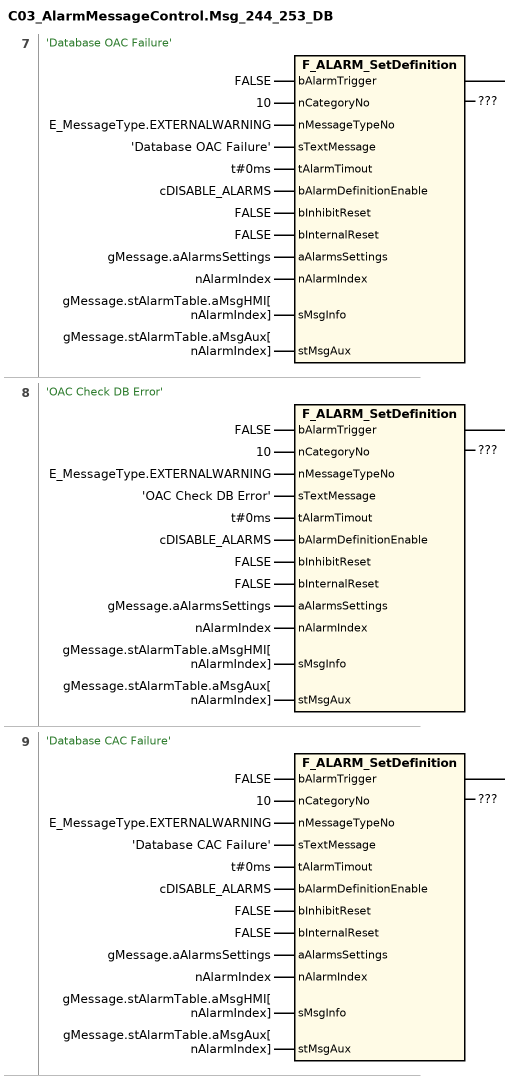
// NETWORK 7
// 'Database OAC Failure'
F_ALARM_SetDefinition(bAlarmTrigger := FALSE, nCategoryNo := 10, nMessageTypeNo := E_MessageType.EXTERNALWARNING, sTextMessage := 'Database OAC Failure', tAlarmTimout := t#0ms, bAlarmDefinitionEnable := cDISABLE_ALARMS, bInhibitReset := FALSE, bInternalReset := FALSE, aAlarmsSettings := gMessage.aAlarmsSettings, nAlarmIndex := nAlarmIndex, sMsgInfo := gMessage.stAlarmTable.aMsgHMI[nAlarmIndex], stMsgAux := gMessage.stAlarmTable.aMsgAux[nAlarmIndex]);

// NETWORK 8
// 'OAC Check DB Error'
F_ALARM_SetDefinition(bAlarmTrigger := FALSE, nCategoryNo := 10, nMessageTypeNo := E_MessageType.EXTERNALWARNING, sTextMessage := 'OAC Check DB Error', tAlarmTimout := t#0ms, bAlarmDefinitionEnable := cDISABLE_ALARMS, bInhibitReset := FALSE, bInternalReset := FALSE, aAlarmsSettings := gMessage.aAlarmsSettings, nAlarmIndex := nAlarmIndex, sMsgInfo := gMessage.stAlarmTable.aMsgHMI[nAlarmIndex], stMsgAux := gMessage.stAlarmTable.aMsgAux[nAlarmIndex]);

// NETWORK 9
// 'Database CAC Failure'
F_ALARM_SetDefinition(bAlarmTrigger := FALSE, nCategoryNo := 10, nMessageTypeNo := E_MessageType.EXTERNALWARNING, sTextMessage := 'Database CAC Failure', tAlarmTimout := t#0ms, bAlarmDefinitionEnable := cDISABLE_ALARMS, bInhibitReset := FALSE, bInternalReset := FALSE, aAlarmsSettings := gMessage.aAlarmsSettings, nAlarmIndex := nAlarmIndex, sMsgInfo := gMessage.stAlarmTable.aMsgHMI[nAlarmIndex], stMsgAux := gMessage.stAlarmTable.aMsgAux[nAlarmIndex]);

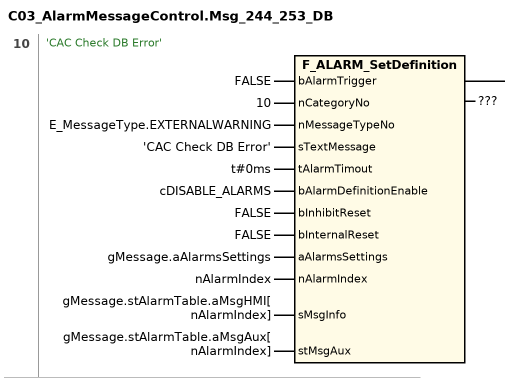
// NETWORK 10
// 'CAC Check DB Error'
F_ALARM_SetDefinition(bAlarmTrigger := FALSE, nCategoryNo := 10, nMessageTypeNo := E_MessageType.EXTERNALWARNING, sTextMessage := 'CAC Check DB Error', tAlarmTimout := t#0ms, bAlarmDefinitionEnable := cDISABLE_ALARMS, bInhibitReset := FALSE, bInternalReset := FALSE, aAlarmsSettings := gMessage.aAlarmsSettings, nAlarmIndex := nAlarmIndex, sMsgInfo := gMessage.stAlarmTable.aMsgHMI[nAlarmIndex], stMsgAux := gMessage.stAlarmTable.aMsgAux[nAlarmIndex]);
END_ACTION

ACTION Msg_254_255_Reserved:
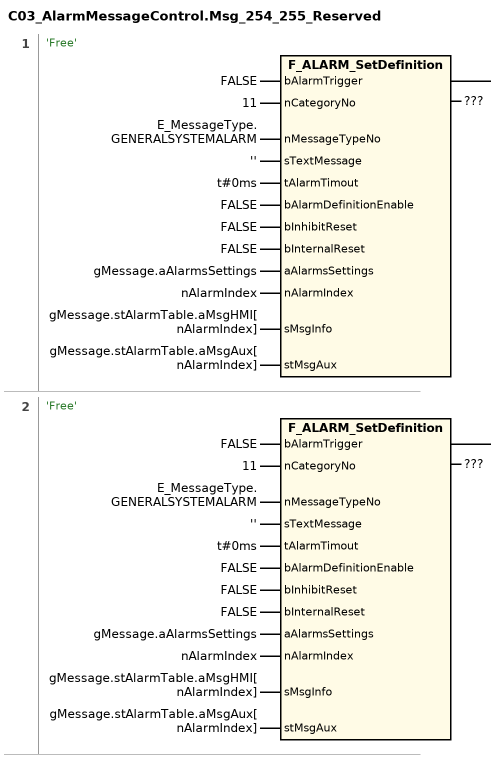
// NETWORK 1
// 'Free'
F_ALARM_SetDefinition(bAlarmTrigger := FALSE, nCategoryNo := 11, nMessageTypeNo := E_MessageType.GENERALSYSTEMALARM, sTextMessage := '', tAlarmTimout := t#0ms, bAlarmDefinitionEnable := FALSE, bInhibitReset := FALSE, bInternalReset := FALSE, aAlarmsSettings := gMessage.aAlarmsSettings, nAlarmIndex := nAlarmIndex, sMsgInfo := gMessage.stAlarmTable.aMsgHMI[nAlarmIndex], stMsgAux := gMessage.stAlarmTable.aMsgAux[nAlarmIndex]);

// NETWORK 2
// 'Free'
F_ALARM_SetDefinition(bAlarmTrigger := FALSE, nCategoryNo := 11, nMessageTypeNo := E_MessageType.GENERALSYSTEMALARM, sTextMessage := '', tAlarmTimout := t#0ms, bAlarmDefinitionEnable := FALSE, bInhibitReset := FALSE, bInternalReset := FALSE, aAlarmsSettings := gMessage.aAlarmsSettings, nAlarmIndex := nAlarmIndex, sMsgInfo := gMessage.stAlarmTable.aMsgHMI[nAlarmIndex], stMsgAux := gMessage.stAlarmTable.aMsgAux[nAlarmIndex]);
END_ACTION

ACTION MsgReset:
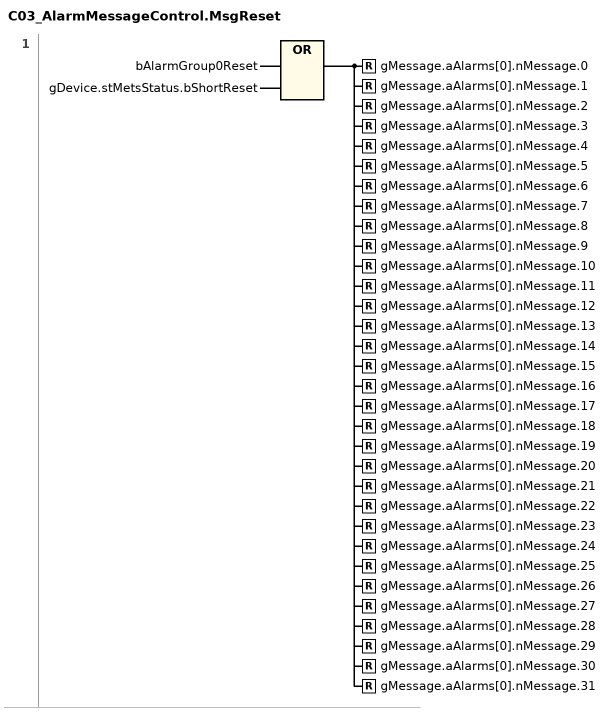
// NETWORK 1
_w1 := bAlarmGroup0Reset OR gDevice.stMetsStatus.bShortReset;
gMessage.aAlarms[0].nMessage.0 R= _w1;
gMessage.aAlarms[0].nMessage.1 R= _w1;
gMessage.aAlarms[0].nMessage.2 R= _w1;
gMessage.aAlarms[0].nMessage.3 R= _w1;
gMessage.aAlarms[0].nMessage.4 R= _w1;
gMessage.aAlarms[0].nMessage.5 R= _w1;
gMessage.aAlarms[0].nMessage.6 R= _w1;
gMessage.aAlarms[0].nMessage.7 R= _w1;
gMessage.aAlarms[0].nMessage.8 R= _w1;
gMessage.aAlarms[0].nMessage.9 R= _w1;
gMessage.aAlarms[0].nMessage.10 R= _w1;
gMessage.aAlarms[0].nMessage.11 R= _w1;
gMessage.aAlarms[0].nMessage.12 R= _w1;
gMessage.aAlarms[0].nMessage.13 R= _w1;
gMessage.aAlarms[0].nMessage.14 R= _w1;
gMessage.aAlarms[0].nMessage.15 R= _w1;
gMessage.aAlarms[0].nMessage.16 R= _w1;
gMessage.aAlarms[0].nMessage.17 R= _w1;
gMessage.aAlarms[0].nMessage.18 R= _w1;
gMessage.aAlarms[0].nMessage.19 R= _w1;
gMessage.aAlarms[0].nMessage.20 R= _w1;
gMessage.aAlarms[0].nMessage.21 R= _w1;
gMessage.aAlarms[0].nMessage.22 R= _w1;
gMessage.aAlarms[0].nMessage.23 R= _w1;
gMessage.aAlarms[0].nMessage.24 R= _w1;
gMessage.aAlarms[0].nMessage.25 R= _w1;
gMessage.aAlarms[0].nMessage.26 R= _w1;
gMessage.aAlarms[0].nMessage.27 R= _w1;
gMessage.aAlarms[0].nMessage.28 R= _w1;
gMessage.aAlarms[0].nMessage.29 R= _w1;
gMessage.aAlarms[0].nMessage.30 R= _w1;
gMessage.aAlarms[0].nMessage.31 R= _w1;

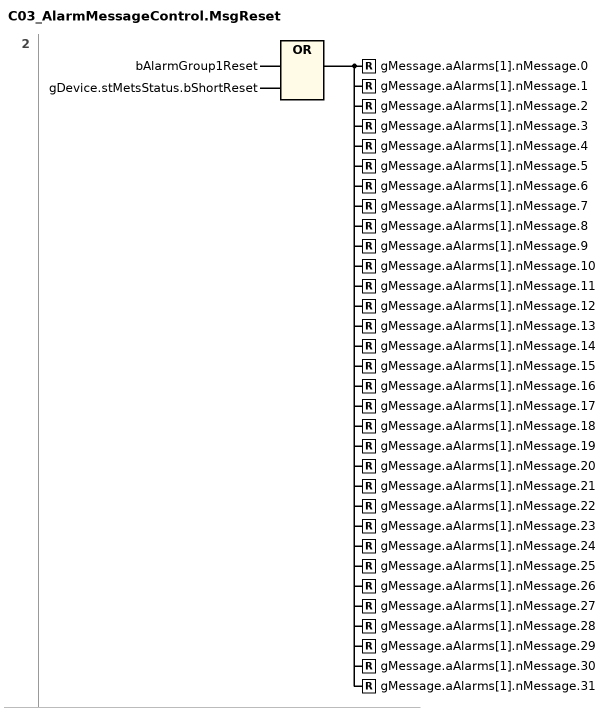
// NETWORK 2
_w2 := bAlarmGroup1Reset OR gDevice.stMetsStatus.bShortReset;
gMessage.aAlarms[1].nMessage.0 R= _w2;
gMessage.aAlarms[1].nMessage.1 R= _w2;
gMessage.aAlarms[1].nMessage.2 R= _w2;
gMessage.aAlarms[1].nMessage.3 R= _w2;
gMessage.aAlarms[1].nMessage.4 R= _w2;
gMessage.aAlarms[1].nMessage.5 R= _w2;
gMessage.aAlarms[1].nMessage.6 R= _w2;
gMessage.aAlarms[1].nMessage.7 R= _w2;
gMessage.aAlarms[1].nMessage.8 R= _w2;
gMessage.aAlarms[1].nMessage.9 R= _w2;
gMessage.aAlarms[1].nMessage.10 R= _w2;
gMessage.aAlarms[1].nMessage.11 R= _w2;
gMessage.aAlarms[1].nMessage.12 R= _w2;
gMessage.aAlarms[1].nMessage.13 R= _w2;
gMessage.aAlarms[1].nMessage.14 R= _w2;
gMessage.aAlarms[1].nMessage.15 R= _w2;
gMessage.aAlarms[1].nMessage.16 R= _w2;
gMessage.aAlarms[1].nMessage.17 R= _w2;
gMessage.aAlarms[1].nMessage.18 R= _w2;
gMessage.aAlarms[1].nMessage.19 R= _w2;
gMessage.aAlarms[1].nMessage.20 R= _w2;
gMessage.aAlarms[1].nMessage.21 R= _w2;
gMessage.aAlarms[1].nMessage.22 R= _w2;
gMessage.aAlarms[1].nMessage.23 R= _w2;
gMessage.aAlarms[1].nMessage.24 R= _w2;
gMessage.aAlarms[1].nMessage.25 R= _w2;
gMessage.aAlarms[1].nMessage.26 R= _w2;
gMessage.aAlarms[1].nMessage.27 R= _w2;
gMessage.aAlarms[1].nMessage.28 R= _w2;
gMessage.aAlarms[1].nMessage.29 R= _w2;
gMessage.aAlarms[1].nMessage.30 R= _w2;
gMessage.aAlarms[1].nMessage.31 R= _w2;

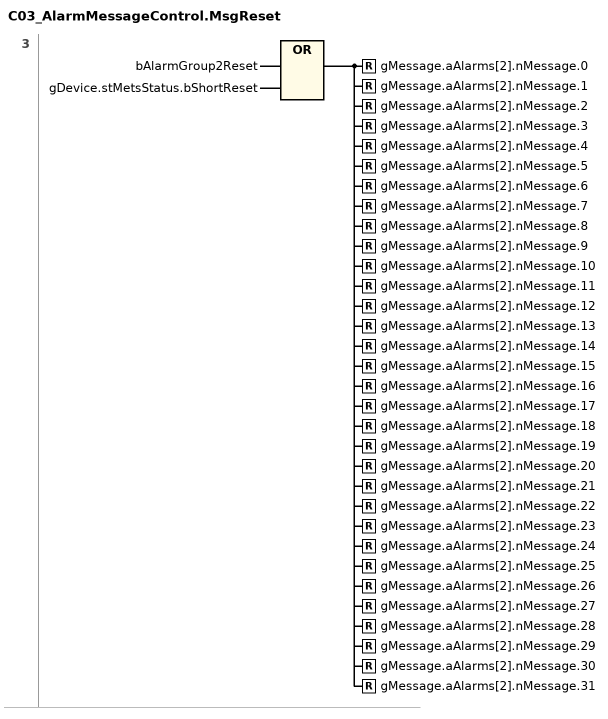
// NETWORK 3
_w3 := bAlarmGroup2Reset OR gDevice.stMetsStatus.bShortReset;
gMessage.aAlarms[2].nMessage.0 R= _w3;
gMessage.aAlarms[2].nMessage.1 R= _w3;
gMessage.aAlarms[2].nMessage.2 R= _w3;
gMessage.aAlarms[2].nMessage.3 R= _w3;
gMessage.aAlarms[2].nMessage.4 R= _w3;
gMessage.aAlarms[2].nMessage.5 R= _w3;
gMessage.aAlarms[2].nMessage.6 R= _w3;
gMessage.aAlarms[2].nMessage.7 R= _w3;
gMessage.aAlarms[2].nMessage.8 R= _w3;
gMessage.aAlarms[2].nMessage.9 R= _w3;
gMessage.aAlarms[2].nMessage.10 R= _w3;
gMessage.aAlarms[2].nMessage.11 R= _w3;
gMessage.aAlarms[2].nMessage.12 R= _w3;
gMessage.aAlarms[2].nMessage.13 R= _w3;
gMessage.aAlarms[2].nMessage.14 R= _w3;
gMessage.aAlarms[2].nMessage.15 R= _w3;
gMessage.aAlarms[2].nMessage.16 R= _w3;
gMessage.aAlarms[2].nMessage.17 R= _w3;
gMessage.aAlarms[2].nMessage.18 R= _w3;
gMessage.aAlarms[2].nMessage.19 R= _w3;
gMessage.aAlarms[2].nMessage.20 R= _w3;
gMessage.aAlarms[2].nMessage.21 R= _w3;
gMessage.aAlarms[2].nMessage.22 R= _w3;
gMessage.aAlarms[2].nMessage.23 R= _w3;
gMessage.aAlarms[2].nMessage.24 R= _w3;
gMessage.aAlarms[2].nMessage.25 R= _w3;
gMessage.aAlarms[2].nMessage.26 R= _w3;
gMessage.aAlarms[2].nMessage.27 R= _w3;
gMessage.aAlarms[2].nMessage.28 R= _w3;
gMessage.aAlarms[2].nMessage.29 R= _w3;
gMessage.aAlarms[2].nMessage.30 R= _w3;
gMessage.aAlarms[2].nMessage.31 R= _w3;

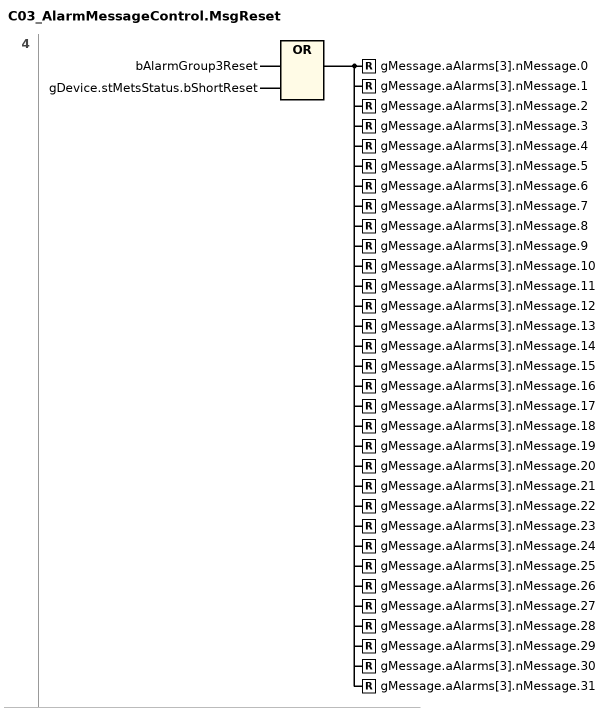
// NETWORK 4
_w4 := bAlarmGroup3Reset OR gDevice.stMetsStatus.bShortReset;
gMessage.aAlarms[3].nMessage.0 R= _w4;
gMessage.aAlarms[3].nMessage.1 R= _w4;
gMessage.aAlarms[3].nMessage.2 R= _w4;
gMessage.aAlarms[3].nMessage.3 R= _w4;
gMessage.aAlarms[3].nMessage.4 R= _w4;
gMessage.aAlarms[3].nMessage.5 R= _w4;
gMessage.aAlarms[3].nMessage.6 R= _w4;
gMessage.aAlarms[3].nMessage.7 R= _w4;
gMessage.aAlarms[3].nMessage.8 R= _w4;
gMessage.aAlarms[3].nMessage.9 R= _w4;
gMessage.aAlarms[3].nMessage.10 R= _w4;
gMessage.aAlarms[3].nMessage.11 R= _w4;
gMessage.aAlarms[3].nMessage.12 R= _w4;
gMessage.aAlarms[3].nMessage.13 R= _w4;
gMessage.aAlarms[3].nMessage.14 R= _w4;
gMessage.aAlarms[3].nMessage.15 R= _w4;
gMessage.aAlarms[3].nMessage.16 R= _w4;
gMessage.aAlarms[3].nMessage.17 R= _w4;
gMessage.aAlarms[3].nMessage.18 R= _w4;
gMessage.aAlarms[3].nMessage.19 R= _w4;
gMessage.aAlarms[3].nMessage.20 R= _w4;
gMessage.aAlarms[3].nMessage.21 R= _w4;
gMessage.aAlarms[3].nMessage.22 R= _w4;
gMessage.aAlarms[3].nMessage.23 R= _w4;
gMessage.aAlarms[3].nMessage.24 R= _w4;
gMessage.aAlarms[3].nMessage.25 R= _w4;
gMessage.aAlarms[3].nMessage.26 R= _w4;
gMessage.aAlarms[3].nMessage.27 R= _w4;
gMessage.aAlarms[3].nMessage.28 R= _w4;
gMessage.aAlarms[3].nMessage.29 R= _w4;
gMessage.aAlarms[3].nMessage.30 R= _w4;
gMessage.aAlarms[3].nMessage.31 R= _w4;

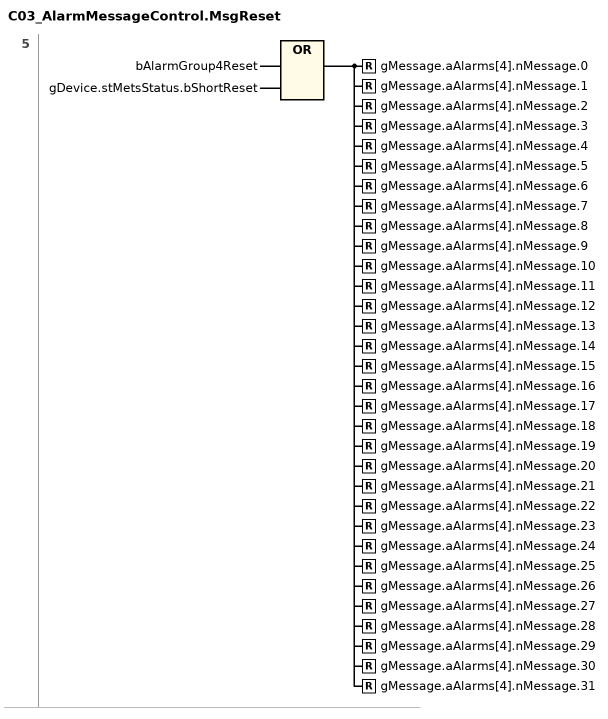
// NETWORK 5
_w5 := bAlarmGroup4Reset OR gDevice.stMetsStatus.bShortReset;
gMessage.aAlarms[4].nMessage.0 R= _w5;
gMessage.aAlarms[4].nMessage.1 R= _w5;
gMessage.aAlarms[4].nMessage.2 R= _w5;
gMessage.aAlarms[4].nMessage.3 R= _w5;
gMessage.aAlarms[4].nMessage.4 R= _w5;
gMessage.aAlarms[4].nMessage.5 R= _w5;
gMessage.aAlarms[4].nMessage.6 R= _w5;
gMessage.aAlarms[4].nMessage.7 R= _w5;
gMessage.aAlarms[4].nMessage.8 R= _w5;
gMessage.aAlarms[4].nMessage.9 R= _w5;
gMessage.aAlarms[4].nMessage.10 R= _w5;
gMessage.aAlarms[4].nMessage.11 R= _w5;
gMessage.aAlarms[4].nMessage.12 R= _w5;
gMessage.aAlarms[4].nMessage.13 R= _w5;
gMessage.aAlarms[4].nMessage.14 R= _w5;
gMessage.aAlarms[4].nMessage.15 R= _w5;
gMessage.aAlarms[4].nMessage.16 R= _w5;
gMessage.aAlarms[4].nMessage.17 R= _w5;
gMessage.aAlarms[4].nMessage.18 R= _w5;
gMessage.aAlarms[4].nMessage.19 R= _w5;
gMessage.aAlarms[4].nMessage.20 R= _w5;
gMessage.aAlarms[4].nMessage.21 R= _w5;
gMessage.aAlarms[4].nMessage.22 R= _w5;
gMessage.aAlarms[4].nMessage.23 R= _w5;
gMessage.aAlarms[4].nMessage.24 R= _w5;
gMessage.aAlarms[4].nMessage.25 R= _w5;
gMessage.aAlarms[4].nMessage.26 R= _w5;
gMessage.aAlarms[4].nMessage.27 R= _w5;
gMessage.aAlarms[4].nMessage.28 R= _w5;
gMessage.aAlarms[4].nMessage.29 R= _w5;
gMessage.aAlarms[4].nMessage.30 R= _w5;
gMessage.aAlarms[4].nMessage.31 R= _w5;

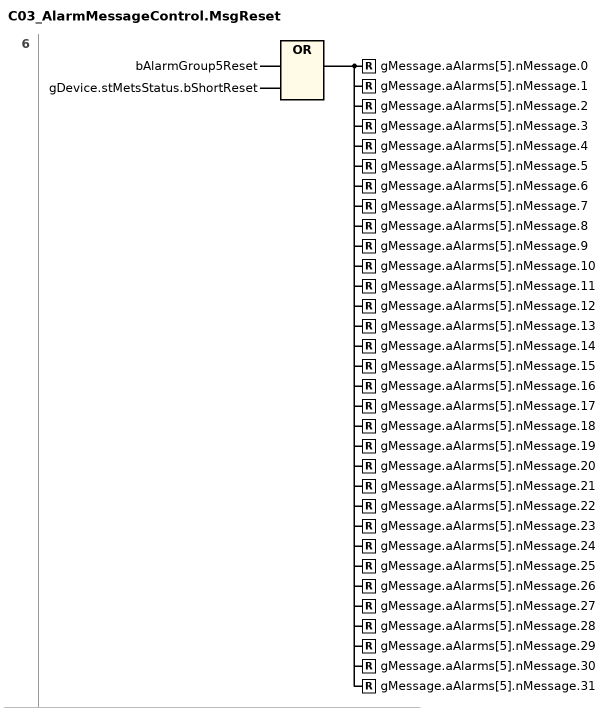
// NETWORK 6
_w6 := bAlarmGroup5Reset OR gDevice.stMetsStatus.bShortReset;
gMessage.aAlarms[5].nMessage.0 R= _w6;
gMessage.aAlarms[5].nMessage.1 R= _w6;
gMessage.aAlarms[5].nMessage.2 R= _w6;
gMessage.aAlarms[5].nMessage.3 R= _w6;
gMessage.aAlarms[5].nMessage.4 R= _w6;
gMessage.aAlarms[5].nMessage.5 R= _w6;
gMessage.aAlarms[5].nMessage.6 R= _w6;
gMessage.aAlarms[5].nMessage.7 R= _w6;
gMessage.aAlarms[5].nMessage.8 R= _w6;
gMessage.aAlarms[5].nMessage.9 R= _w6;
gMessage.aAlarms[5].nMessage.10 R= _w6;
gMessage.aAlarms[5].nMessage.11 R= _w6;
gMessage.aAlarms[5].nMessage.12 R= _w6;
gMessage.aAlarms[5].nMessage.13 R= _w6;
gMessage.aAlarms[5].nMessage.14 R= _w6;
gMessage.aAlarms[5].nMessage.15 R= _w6;
gMessage.aAlarms[5].nMessage.16 R= _w6;
gMessage.aAlarms[5].nMessage.17 R= _w6;
gMessage.aAlarms[5].nMessage.18 R= _w6;
gMessage.aAlarms[5].nMessage.19 R= _w6;
gMessage.aAlarms[5].nMessage.20 R= _w6;
gMessage.aAlarms[5].nMessage.21 R= _w6;
gMessage.aAlarms[5].nMessage.22 R= _w6;
gMessage.aAlarms[5].nMessage.23 R= _w6;
gMessage.aAlarms[5].nMessage.24 R= _w6;
gMessage.aAlarms[5].nMessage.25 R= _w6;
gMessage.aAlarms[5].nMessage.26 R= _w6;
gMessage.aAlarms[5].nMessage.27 R= _w6;
gMessage.aAlarms[5].nMessage.28 R= _w6;
gMessage.aAlarms[5].nMessage.29 R= _w6;
gMessage.aAlarms[5].nMessage.30 R= _w6;
gMessage.aAlarms[5].nMessage.31 R= _w6;

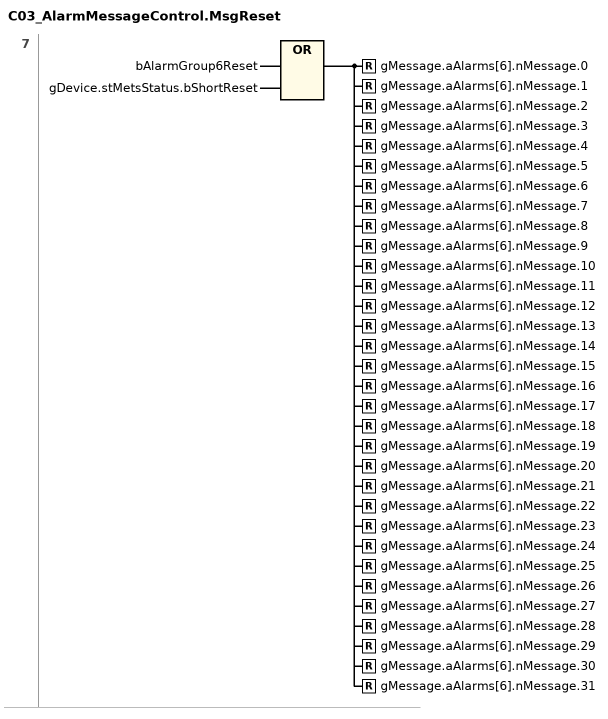
// NETWORK 7
_w7 := bAlarmGroup6Reset OR gDevice.stMetsStatus.bShortReset;
gMessage.aAlarms[6].nMessage.0 R= _w7;
gMessage.aAlarms[6].nMessage.1 R= _w7;
gMessage.aAlarms[6].nMessage.2 R= _w7;
gMessage.aAlarms[6].nMessage.3 R= _w7;
gMessage.aAlarms[6].nMessage.4 R= _w7;
gMessage.aAlarms[6].nMessage.5 R= _w7;
gMessage.aAlarms[6].nMessage.6 R= _w7;
gMessage.aAlarms[6].nMessage.7 R= _w7;
gMessage.aAlarms[6].nMessage.8 R= _w7;
gMessage.aAlarms[6].nMessage.9 R= _w7;
gMessage.aAlarms[6].nMessage.10 R= _w7;
gMessage.aAlarms[6].nMessage.11 R= _w7;
gMessage.aAlarms[6].nMessage.12 R= _w7;
gMessage.aAlarms[6].nMessage.13 R= _w7;
gMessage.aAlarms[6].nMessage.14 R= _w7;
gMessage.aAlarms[6].nMessage.15 R= _w7;
gMessage.aAlarms[6].nMessage.16 R= _w7;
gMessage.aAlarms[6].nMessage.17 R= _w7;
gMessage.aAlarms[6].nMessage.18 R= _w7;
gMessage.aAlarms[6].nMessage.19 R= _w7;
gMessage.aAlarms[6].nMessage.20 R= _w7;
gMessage.aAlarms[6].nMessage.21 R= _w7;
gMessage.aAlarms[6].nMessage.22 R= _w7;
gMessage.aAlarms[6].nMessage.23 R= _w7;
gMessage.aAlarms[6].nMessage.24 R= _w7;
gMessage.aAlarms[6].nMessage.25 R= _w7;
gMessage.aAlarms[6].nMessage.26 R= _w7;
gMessage.aAlarms[6].nMessage.27 R= _w7;
gMessage.aAlarms[6].nMessage.28 R= _w7;
gMessage.aAlarms[6].nMessage.29 R= _w7;
gMessage.aAlarms[6].nMessage.30 R= _w7;
gMessage.aAlarms[6].nMessage.31 R= _w7;

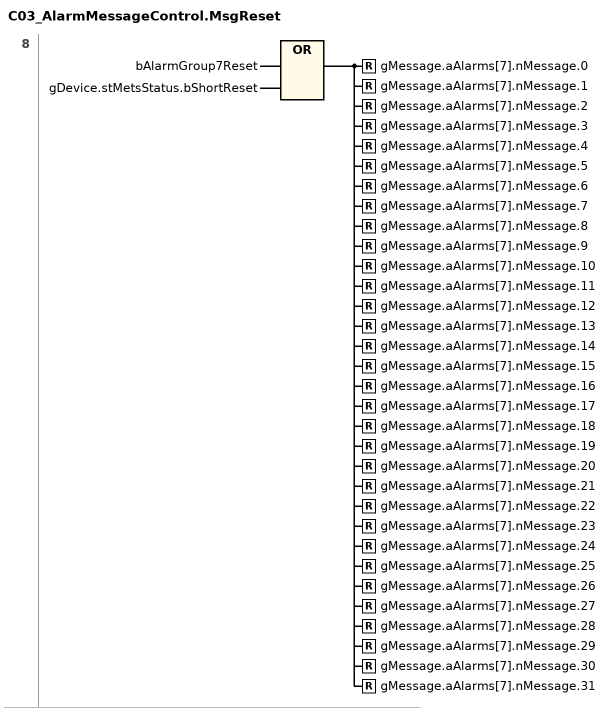
// NETWORK 8
_w8 := bAlarmGroup7Reset OR gDevice.stMetsStatus.bShortReset;
gMessage.aAlarms[7].nMessage.0 R= _w8;
gMessage.aAlarms[7].nMessage.1 R= _w8;
gMessage.aAlarms[7].nMessage.2 R= _w8;
gMessage.aAlarms[7].nMessage.3 R= _w8;
gMessage.aAlarms[7].nMessage.4 R= _w8;
gMessage.aAlarms[7].nMessage.5 R= _w8;
gMessage.aAlarms[7].nMessage.6 R= _w8;
gMessage.aAlarms[7].nMessage.7 R= _w8;
gMessage.aAlarms[7].nMessage.8 R= _w8;
gMessage.aAlarms[7].nMessage.9 R= _w8;
gMessage.aAlarms[7].nMessage.10 R= _w8;
gMessage.aAlarms[7].nMessage.11 R= _w8;
gMessage.aAlarms[7].nMessage.12 R= _w8;
gMessage.aAlarms[7].nMessage.13 R= _w8;
gMessage.aAlarms[7].nMessage.14 R= _w8;
gMessage.aAlarms[7].nMessage.15 R= _w8;
gMessage.aAlarms[7].nMessage.16 R= _w8;
gMessage.aAlarms[7].nMessage.17 R= _w8;
gMessage.aAlarms[7].nMessage.18 R= _w8;
gMessage.aAlarms[7].nMessage.19 R= _w8;
gMessage.aAlarms[7].nMessage.20 R= _w8;
gMessage.aAlarms[7].nMessage.21 R= _w8;
gMessage.aAlarms[7].nMessage.22 R= _w8;
gMessage.aAlarms[7].nMessage.23 R= _w8;
gMessage.aAlarms[7].nMessage.24 R= _w8;
gMessage.aAlarms[7].nMessage.25 R= _w8;
gMessage.aAlarms[7].nMessage.26 R= _w8;
gMessage.aAlarms[7].nMessage.27 R= _w8;
gMessage.aAlarms[7].nMessage.28 R= _w8;
gMessage.aAlarms[7].nMessage.29 R= _w8;
gMessage.aAlarms[7].nMessage.30 R= _w8;
gMessage.aAlarms[7].nMessage.31 R= _w8;
END_ACTION

END_PROGRAM

(* stored: Version 1.1.0.1
   POU C03_AlarmMessageControl: Id {08bc1f85-53a7-41a4-86b5-45f09ed07d2c}, SpecialFunc None
   Action Msg_000_033_General: Id {33e6d5ff-68f1-435c-bdf8-00050c4b0ba0}
   Action Msg_034_074_Cameras: Id {3a5dbdb5-da2c-400a-8cf9-cd3a2340a6bd}
   Action Msg_075_126_Process: Id {59597455-697b-455d-92d5-d61434209beb}
   Action Msg_127_150_Sensors: Id {231a3438-1136-4452-9624-eab1da84a3f7}
   Action Msg_151_179_Doors: Id {7dc34f72-21b8-4ff7-85a8-315f3873c80e}
   Action Msg_180_200_Motors: Id {4b49261a-c499-452d-8cca-d8389d7b9fc8}
   Action Msg_201_208_Interface: Id {7e7d6b6b-49a3-4fe5-b188-375f1f755118}
   Action Msg_209_237_Labellers: Id {ed72f88d-e679-4f21-b51b-79e4e4393ee4}
   Action Msg_238_243_Spare: Id {f803fcc3-d030-4940-9c39-5d23c0390d0b}
   Action Msg_244_253_DB: Id {81aec2ca-ded1-453f-abe5-f369b4c8b400}
   Action Msg_254_255_Reserved: Id {cb97a817-db56-4447-99e0-fef9c7b60e64}
   Action MsgReset: Id {57fca57a-c51f-49bf-8294-1ad076ee3d78} *)
